// Mitsubishi GX Works2 project: 실수를 정수로   PLC: Q02/Q02H

PROGRAM MAIN
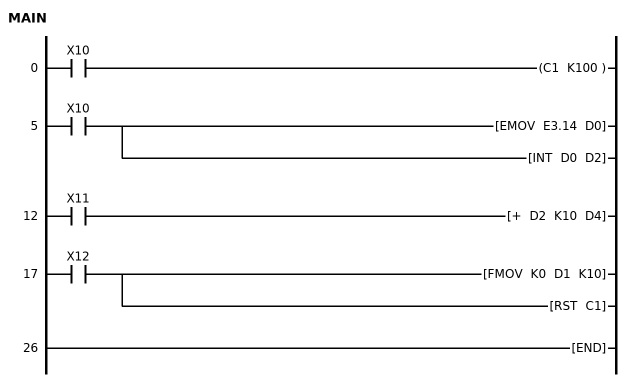
0     LD      X10
      OUT     C1 K100
5     LD      X10
      EMOV    E3.14 D0
      INT     D0 D2
12    LD      X11
      +       D2 K10 D4
17    LD      X12
      FMOV    K0 D1 K10
      RST     C1
26    END
END_PROGRAM
